FUNCTION_BLOCK FB_RollingAverageConsumer
VAR
    adder : B1RollingAverage_Plc.FB_RollingAverage;
    lastResult : INT;
END_VAR

lastResult := adder.Step(sample := 10);

END_FUNCTION_BLOCK

(* stored: Version 1.1.0.1
   POU FB_RollingAverageConsumer: Id {e49e35ac-14b7-437c-b940-efd19e3c0caf}, SpecialFunc None *)
